PROGRAM MAIN_2
VAR
	counter_2:INT:=0;
END_VAR

counter_2:=counter_2+1;

END_PROGRAM

(* stored: Version 1.1.0.1, ProductVersion 3.1.4024.9
   POU MAIN_2: Id {c42b9b1e-d303-4193-95be-85832af438f4}, SpecialFunc None *)
